// TIA Portal project "Ass 2" (V15)

(* hardware
DEVICE "S7-1200 station_1"  S7-1200 Station
   slot 0: "Rack_0"  S7-1200 Rack  Rack  V1.0
   slot 1: "PLC_1"  CPU 1215C AC/DC/Rly  6ES7 215-1BG40-0XB0  V4.0
*)

// ===== PLC "PLC_1"  CPU 1215C AC/DC/Rly =====

VAR_GLOBAL   // PLC tag table "Vari"
   "Start/Stop" AT %M0.0 : Bool;
   "Stop" AT %M0.1 : Bool;
   "Tank B Level Scaled" AT %QD16 : Real;
   "Tank Level Difference" AT %QD20 : Real;
   "Tank Level Difference ABS" AT %QD24 : Real;
   "Pump 1" AT %Q0.4 : Bool;
   "Pump 2" AT %Q0.5 : Bool;
   "Tank A Level" AT %MW64 : Word;
   "Tank B Level" AT %MW66 : Word;
   "Tank A Level Norm" AT %QD2 : Real;
   "Tank B Level Norm" AT %QD6 : Real;
   "Tank A Level Scaled" AT %QD10 : Real;
   "Tank A" AT %Q0.6 : Bool;
   "Tank B" AT %Q0.7 : Bool;
END_VAR

// folder: System blocks/Program resources

DATA_BLOCK "IEC_Timer_0_DB"   // DB1
{ S7_Optimized_Access := 'TRUE' }
AUTHOR : Simatic
FAMILY : IEC
NAME : IEC_TMR
VERSION : 1.0
// stored: InstanceOfName IEC_TIMER
"IEC_TIMER"
BEGIN
END_DATA_BLOCK

DATA_BLOCK "IEC_Timer_0_DB_1"   // DB2
{ S7_Optimized_Access := 'TRUE' }
AUTHOR : Simatic
FAMILY : IEC
NAME : IEC_TMR
VERSION : 1.0
// stored: InstanceOfName IEC_TIMER
"IEC_TIMER"
BEGIN
END_DATA_BLOCK

// folder: (top level)

ORGANIZATION_BLOCK "Main"   // OB1, LAD, ProgramCycle
TITLE = "Main Program Sweep (Cycle)"
{ S7_Optimized_Access := 'TRUE' }
VERSION : 0.1
// Cascade Tank Level Equalization
// 
// Objective: Maintain two tanks at roughly the same level.
// Required: Scale both tank levels (0-100%). 
// Use Arithmetic to find the absolute difference: Tank A  Tank B (using ABS function if available, or just subtract both ways). 
// Use Comparators to open a transfer pump if the difference > 20%. 
// Use a Timer (10 seconds) to delay the pump start to prevent chasing minor fluctuations
   VAR_INPUT
      Initial_Call : Bool;   // Initial call of this OB
      Remanence : Bool;   // =True, if remanent data are available
   END_VAR
BEGIN

REGION Network 1
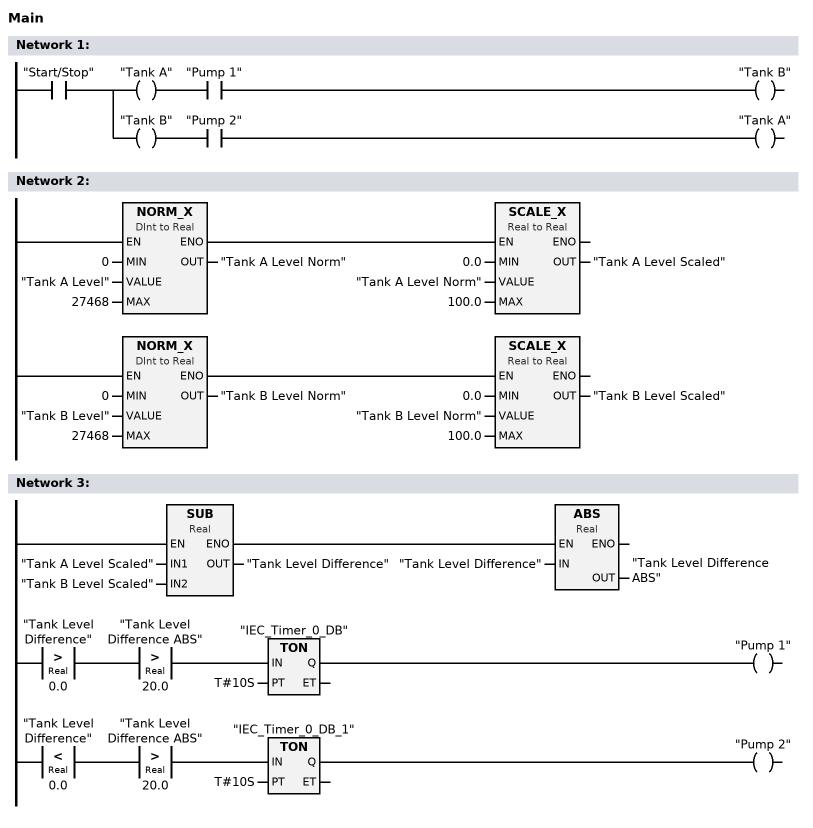
   RUNG wire#powerrail
      Contact( "Start/Stop" )
      wire#w1
      Coil( "Tank A" )
      Contact( "Pump 1" )
      Coil( "Tank B" )
   END_RUNG
   RUNG wire#w1
      Coil( "Tank B" )
      Contact( "Pump 2" )
      Coil( "Tank A" )
   END_RUNG
   // the same network as SCL:
   "Tank A" := "Start/Stop";
   "Tank B" := "Start/Stop" AND "Pump 1";
   "Tank B" := "Start/Stop";
   "Tank A" := "Start/Stop" AND "Pump 2";
END_REGION

REGION Network 2
   RUNG wire#powerrail
      { S7_Templates := "[SrcType := DInt, DestType := Real]" } Normalize(min := 0, value := "Tank A Level", max := 27468, out => "Tank A Level Norm")
      { S7_Templates := "[SrcType := Real, DestType := Real]" } Scale(min := 0.0, value := "Tank A Level Norm", max := 100.0, out => "Tank A Level Scaled")
   END_RUNG
   RUNG wire#powerrail
      { S7_Templates := "[SrcType := DInt, DestType := Real]" } Normalize(min := 0, value := "Tank B Level", max := 27468, out => "Tank B Level Norm")
      { S7_Templates := "[SrcType := Real, DestType := Real]" } Scale(min := 0.0, value := "Tank B Level Norm", max := 100.0, out => "Tank B Level Scaled")
   END_RUNG
   // the same network as SCL:
   "Tank A Level Norm" := NORM_X(MIN := 0, VALUE := "Tank A Level", MAX := 27468);
   "Tank A Level Scaled" := SCALE_X(MIN := 0.0, VALUE := "Tank A Level Norm", MAX := 100.0);
   "Tank B Level Norm" := NORM_X(MIN := 0, VALUE := "Tank B Level", MAX := 27468);
   "Tank B Level Scaled" := SCALE_X(MIN := 0.0, VALUE := "Tank B Level Norm", MAX := 100.0);
END_REGION

REGION Network 3
   "Tank Level Difference" := "Tank A Level Scaled" - "Tank B Level Scaled";
   "Tank Level Difference ABS" := ABS("Tank Level Difference");
   "IEC_Timer_0_DB".TON(IN := ("Tank Level Difference" > 0.0) AND ("Tank Level Difference ABS" > 20.0),
                        PT := T#10S);
   "Pump 1" := "IEC_Timer_0_DB".Q;
   "IEC_Timer_0_DB_1".TON(IN := ("Tank Level Difference" < 0.0) AND ("Tank Level Difference ABS" > 20.0),
                          PT := T#10S);
   "Pump 2" := "IEC_Timer_0_DB_1".Q;
END_REGION
END_ORGANIZATION_BLOCK